{attribute 'qualified_only'}
VAR_GLOBAL
	
	tDelay					:TIME:= T#1S;
	
	//=====================UI Button=============================
	bStartBtnUI			:BOOL;	(*butto from UI*)
	bStopBtnUI			:BOOL;	(*butto from UI*)
	bPauseBtnUI			:BOOL;	(*butto from UI*)
	//=====================UI Button=============================
	
	btemp		:BOOL;
	
	//=============Function Blcok instance===================
	fbMarqueeExPause		:FB_MarqueeExPause:=(pLamp01:=ADR(GVL_Machine.HWIO.HWOutput.Lamp01),pLamp02:=ADR(GVL_Machine.HWIO.HWOutput.Lamp02),
												pLamp03:=ADR(GVL_Machine.HWIO.HWOutput.Lamp03),pLamp04:=ADR(GVL_Machine.HWIO.HWOutput.Lamp04),
												pTime:=ADR(GVL_General.tDelay),
												pPause:=ADR(GVL_SignalHanlding.inPauseBtnHandling.bSignalOutput),														
												pStop:=ADR(GVL_SignalHanlding.inStopBtnHandling.bSignalOutput));
	
	
	
END_VAR

(* stored: Version 1.1.0.1, ProductVersion 3.1.4022.16
   GVL GVL_General: Id {be71a7b4-7ff8-4846-af8b-dba340512ccd} *)
